FUNCTION_BLOCK FB_Object
VAR_INPUT
END_VAR
VAR_OUTPUT
END_VAR
VAR
	iMem:UINT;
END_VAR

METHOD PUBLIC M_Add : UINT
VAR_INPUT
	iVal:UINT;
END_VAR
iMem:=iMem+iVal;
M_Add:=iMem;
END_METHOD

PROPERTY PUBLIC P_Memory : uint
GET
P_Memory:=iMem;
END_GET
SET
iMem:=P_Memory;
END_SET
END_PROPERTY

END_FUNCTION_BLOCK

(* stored: Version 1.1.0.1, ProductVersion 3.1.4024.2
   POU FB_Object: Id {70c817b1-e61c-405f-8420-4660f29a259c}, SpecialFunc None
   Method M_Add: Id {986fa425-7676-40fd-8946-3e70a8c7dfc5}
   Property P_Memory: Id {d36105d0-f554-45c5-84cf-081f7f04df7f}
   Get Get: Id {78e6aa4b-0dcf-46a5-95f2-d65bdd885daa}
   Set Set: Id {51784b65-e8f8-40aa-8cf8-9aeb1a4b137e} *)
